// TIA Portal V15 export
// export: Created 2018-12-10T18:36:36.3562855Z, ExportSetting WithDefaults, WithReadOnly, DisplayName Totally Integrated Automation Portal, DisplayVersion V15 Update 2, DisplayName TIA Portal Openness, DisplayVersion V15 Update 2, DisplayName STEP 7 Professional, DisplayVersion V15 Update 2, DisplayName STEP 7 Safety, DisplayVersion V15, DisplayName WinCC Professional, DisplayVersion V15 Update 2, DisplayName SIMATIC Visualization Architect, DisplayVersion V15 Update 1
FUNCTION "FIXTURENAME_Call" : Void   // FC41, FBD
TITLE = FIXTURENAME Geo station / FIXTURENAME Geostation
{ S7_Optimized_Access := 'FALSE' }
VERSION : 0.1
// stored: AutoNumber true, CodeModifiedDate 2018-01-29T16:41:53.1247001Z, CompileDate 2018-02-20T10:24:53.3770226Z, CreationDate 2016-05-26T15:12:40.5479205Z, HandleErrorsWithinBlock false, InterfaceModifiedDate 2017-10-27T11:23:28.0041837Z, IsConsistent true, IsIECCheckEnabled false, IsKnowHowProtected false, IsWriteProtected false, LibraryConformanceStatus The object is library-conformant., ModifiedDate 2018-01-29T16:41:53.1247001Z, ParameterModified 2017-10-27T11:23:27.956181Z, PLCSimAdvancedSupport false, SetENOAutomatically False, StructureModified 2017-10-27T11:23:28.0041837Z, UDAEnableTagReadback false
BEGIN
END_FUNCTION
